{attribute 'GeneratedUsingTerminal: ATH2000-5250-0022'}
{attribute addProperty BoxType "ATH2000-5250-0022"}
{attribute addProperty Description "ATH2000-5250 Hygienic Sensor line"}
{attribute addProperty Physics "K"}
{attribute addProperty Id "FB_InputsAT %I*FB_Inputs_2D6658510FB_OutputsAT %Q*FB_Outputs_DAFD38E02WcStateAT %I*WcState_9091E0EB2InfoDataAT %I*InfoData_A7436BC610"}
{attribute addProperty CRC "3631482894"}
{attribute addProperty Size "14"}
TYPE ATH2000_D874080E EXTENDS EtcSlaveTerminalBase_947E5A46 :
STRUCT
	{attribute addProperty Name "FB_Inputs"}
	FB_Inputs : FB_Inputs_2D665851;
	{attribute addProperty Name "FB_Outputs"}
	FB_Outputs : FB_Outputs_DAFD38E0;
	{attribute addProperty Name "WcState"}
	WcState : WcState_9091E0EB;
	{attribute addProperty Name "InfoData"}
	InfoData : InfoData_A7436BC6;
END_STRUCT
END_TYPE

(* stored: Version 1.2.0.0, ProductVersion 3.1.4024.11
   DUT ATH2000_D874080E: Id {40eb8299-f712-47ff-83c5-d1cf307689e1} *)
